FUNCTION Convert_DWORD_TO_DT : Hresult
VAR_INPUT
	in : DWORD;
	out : REFERENCE TO DT;
END_VAR
VAR
	converted : DT;
END_VAR

converted := DWORD_TO_DT(in);

IF (DT_TO_DWORD(converted) <> in) THEN
	Convert_DWORD_TO_DT := INCOMPATIBLE;
	RETURN;
END_IF

out := converted;

END_FUNCTION

(* stored: Version 1.1.0.1, ProductVersion 3.1.4024.12
   POU Convert_DWORD_TO_DT: Id {c279c4bd-81e9-4e6a-bae0-d41c9d9a8e4a}, SpecialFunc None *)
